FUNCTION_BLOCK E_TABLE (* Composite Function Block Type *)
  (* Standard: 61499-1 Annex A; Description: Copyright (c) 2017 fortiss GmbH This program and the accompanying materials are made available under the terms of the Eclipse Public License 2.0 which is available at https://www.eclipse.org/legal/epl-2.0/ SPDX-License-Identifier: EPL-2.0 *)
  (* Version 1.0, 2017-09-22, Alois Zoitl, fortiss GmbH, initial API and implementation and/or initial documentation *)
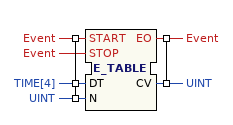
  EVENT_INPUT
    START WITH DT, N; (* Start table driven event generation *)
    STOP; (* Stop table driven event generation *)
  END_EVENT
  EVENT_OUTPUT
    EO WITH CV; (* Generated events *)
  END_EVENT
  VAR_INPUT
    DT : ARRAY [0..3] OF TIME;
    N : UINT;
  END_VAR
  VAR_OUTPUT
    CV : UINT;
  END_VAR
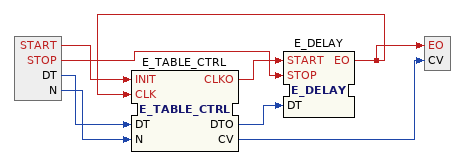
  FBS
    E_TABLE_CTRL : E_TABLE_CTRL;
    E_DELAY : E_DELAY;
  END_FBS
  EVENT_CONNECTIONS
    E_TABLE_CTRL.CLKO TO E_DELAY.START;
    E_DELAY.EO TO EO;
    START TO E_TABLE_CTRL.INIT;
    E_DELAY.EO TO E_TABLE_CTRL.CLK;
    STOP TO E_DELAY.STOP;
  END_CONNECTIONS
  DATA_CONNECTIONS
    E_TABLE_CTRL.DTO TO E_DELAY.DT;
    E_TABLE_CTRL.CV TO CV;
    DT TO E_TABLE_CTRL.DT;
    N TO E_TABLE_CTRL.N;
  END_CONNECTIONS
END_FUNCTION_BLOCK
